FUNCTION_BLOCK SimpleLogMessage IMPLEMENTS I_SimpleLogMessage
VAR
	{attribute 'hide'}
	_Message : T_MaxString;
	{attribute 'hide'}
	_Severity : USINT;
END_VAR

{attribute 'monitoring' := 'call'}
PROPERTY Message : T_MaxString
GET
Message := _Message;
END_GET
SET
_Message := Message;
END_SET
END_PROPERTY

{attribute 'monitoring' := 'call'}
PROPERTY Severity : USINT
GET
Severity := _Severity;
END_GET
SET
_Severity := Severity;
END_SET
END_PROPERTY

END_FUNCTION_BLOCK

(* stored: Version 1.1.0.1
   POU SimpleLogMessage: Id {e5e6ec48-28df-4f2e-ae31-0ae077ba406e}, SpecialFunc None
   Property Message: Id {49a69073-4b54-4d5d-8ded-7b644c92f604}
   Get Get: Id {86617bc2-1b08-4d06-aaaf-7bb478b3c7fe}
   Set Set: Id {496e07a1-59d2-45d0-8b42-f4e5bc9da1aa}
   Property Severity: Id {d3679c17-7738-4898-b01f-a6d741b33dce}
   Get Get: Id {6aa8816a-3ef8-4d31-af8a-f7ce3940f786}
   Set Set: Id {fc63e5a8-aac9-4b68-ae59-d1dfadaa8148} *)
